// TIA Portal V15.1 export
// export: Created 2024-06-21T08:41:06.2222492Z, ExportSetting WithDefaults, DisplayName Totally Integrated Automation Portal, DisplayVersion V15.1 Update 5, DisplayName TIA Portal Openness, DisplayVersion V15.1 Update 5, DisplayName SINAMICS Startdrive Advanced, DisplayVersion V15.1, DisplayName G130, G150, S120, S150, SINAMICS MV, S210, DisplayVersion V15.1, DisplayName G110M, G120, G120C, G120D, G120P, DisplayVersion V15.1, DisplayName STEP 7 Professional, DisplayVersion V15.1 Update 5, DisplayName STEP 7 Safety, DisplayVersion V15.1, DisplayName WinCC Professional, DisplayVersion V15.1 Update 5, DisplayName SIMATIC Visualization Architect, DisplayVersion V15.1
FUNCTION_BLOCK "LGBMotorEPos-MoviProPN"   // FB6622, FBD
TITLE = LMotorMovUnitEPos-MoviProPN / LGBMotorEPos-MoviProPN
{ S7_Optimized_Access := 'TRUE' }
VERSION : 0.1
// ============================================================================
// This module is used in applications when a Motor positioning equipped with SEW MOVIPRO with fieldbus steering is needed.
// ============================================================================
// stored: AutoNumber false, IsIECCheckEnabled false, IsRetainMemResEnabled false, MemoryReserve 100, SetENOAutomatically False, UDAEnableTagReadback false
   VAR_INPUT
      I_MotorProtection { ExternalAccessible := 'False'; ExternalVisible := 'False'; ExternalWritable := 'False'} : Bool;   // Motor protection
      I_AlarmResetPB { ExternalAccessible := 'False'; ExternalVisible := 'False'; ExternalWritable := 'False'} : Bool;   // Alarm Reset Pushbutton is Activated
      I_SafetyStatusWord { ExternalAccessible := 'False'; ExternalVisible := 'False'; ExternalWritable := 'False'} : Word;   // Safety status word
      I_SafetyControlWord { ExternalAccessible := 'False'; ExternalVisible := 'False'; ExternalWritable := 'False'} : Word;   // Safety control word
      I_SafetyOk { ExternalAccessible := 'False'; ExternalVisible := 'False'; ExternalWritable := 'False'} : Bool;   // Safety ok
      I_MotionStopOk { ExternalAccessible := 'False'; ExternalVisible := 'False'; ExternalWritable := 'False'} : Bool;   // Safety Ok / The motion stop is Ok
      I_ContolInhibit { ExternalAccessible := 'False'; ExternalVisible := 'False'; ExternalWritable := 'False'} : Bool;   // Inhibit motor (disable output stage, uncontolled stop)
      I_Start { ExternalAccessible := 'False'; ExternalVisible := 'False'; ExternalWritable := 'False'} : Bool;
      I_OFF2 { ExternalAccessible := 'False'; ExternalVisible := 'False'; ExternalWritable := 'False'} : Bool := True;   // OFF2 rapid stop
      I_SetpointPosition { ExternalAccessible := 'False'; ExternalVisible := 'False'; ExternalWritable := 'False'} : DInt;   // Setpoint position [ user unit ex: rev. ]
      I_SetpointSpeed { ExternalAccessible := 'False'; ExternalVisible := 'False'; ExternalWritable := 'False'} : Int;   // Setpoint velocity [ user unit ex: rev./min ]
      I_Acceleration { ExternalAccessible := 'False'; ExternalVisible := 'False'; ExternalWritable := 'False'} : Int;   // Acceleration [ user unit ex: rev./(min*S) ]
      I_Deceleration { ExternalAccessible := 'False'; ExternalVisible := 'False'; ExternalWritable := 'False'} : Int;   // Deceleration [ user unit ex: rev./(min*S) ]
      I_OperatingMode { ExternalAccessible := 'False'; ExternalVisible := 'False'; ExternalWritable := 'False'} : USInt := 4;   // 0=Default, 1=Speed control, 2=Jog mode, 3=Referencing mode, 4=Positioning mode, 5=Positioning mode - touch probe, 6=Speed synchronization, 7=Emergency mode
      I_BrakeRelease { ExternalAccessible := 'False'; ExternalVisible := 'False'; ExternalWritable := 'False'} : Bool;   // Command brake release
      I_DisableSoftwareLimitSwitches { ExternalAccessible := 'False'; ExternalVisible := 'False'; ExternalWritable := 'False'} : Bool;   // Disable softwrare limit switches in the drive
      I_EnableTorqueLimiting { ExternalAccessible := 'False'; ExternalVisible := 'False'; ExternalWritable := 'False'} : Bool;   // Enable torque limiting
      I_JogPositive { ExternalAccessible := 'False'; ExternalVisible := 'False'; ExternalWritable := 'False'} : Bool;   // Jog in positive direction
      I_JogNegative { ExternalAccessible := 'False'; ExternalVisible := 'False'; ExternalWritable := 'False'} : Bool;   // Jog in negative direction
   END_VAR
   VAR_OUTPUT
      O_MotorProtectionAlarm { ExternalAccessible := 'False'; ExternalVisible := 'False'; ExternalWritable := 'False'} : Bool;   // Motor protection alarm
      O_SafetySwitchAlarm { ExternalAccessible := 'False'; ExternalVisible := 'False'; ExternalWritable := 'False'} : Bool;   // Safety switch alarm
      O_STOAlarm { ExternalAccessible := 'False'; ExternalVisible := 'False'; ExternalWritable := 'False'} : Bool;   // Drive fault / STO alarm
      O_MotionStopWarning { ExternalAccessible := 'False'; ExternalVisible := 'False'; ExternalWritable := 'False'} : Bool;   // Drive fault / Motion Stop warning
      O_DriveFaultAlarm { ExternalAccessible := 'False'; ExternalVisible := 'False'; ExternalWritable := 'False'} : Bool;   // Drive fault
      O_DriveWarning { ExternalAccessible := 'False'; ExternalVisible := 'False'; ExternalWritable := 'False'} : Bool;   // Drive warning
      O_DriveReady { ExternalAccessible := 'False'; ExternalVisible := 'False'; ExternalWritable := 'False'} : Bool;   // Drive ready
      O_Referenced { ExternalAccessible := 'False'; ExternalVisible := 'False'; ExternalWritable := 'False'} : Bool;   // Drive is referenced
      O_MotorTurning { ExternalAccessible := 'False'; ExternalVisible := 'False'; ExternalWritable := 'False'} : Bool;   // Inverter output stage is enabled
      O_Brake { ExternalAccessible := 'False'; ExternalVisible := 'False'; ExternalWritable := 'False'} : Bool;   // Brake status
      O_Standstill { ExternalAccessible := 'False'; ExternalVisible := 'False'; ExternalWritable := 'False'} : Bool;   // Sandstill
      O_SetpointReached { ExternalAccessible := 'False'; ExternalVisible := 'False'; ExternalWritable := 'False'} : Bool;   // Setpoint position is reached
      O_HWLSPositive { ExternalAccessible := 'False'; ExternalVisible := 'False'; ExternalWritable := 'False'} : Bool;   // Hardware limit switch positive reached
      O_HWLSNegative { ExternalAccessible := 'False'; ExternalVisible := 'False'; ExternalWritable := 'False'} : Bool;   // Hardware limit switch negative reached
      O_NoResponse { ExternalAccessible := 'False'; ExternalVisible := 'False'; ExternalWritable := 'False'} : Bool;   // No response / O_NoResponse
      O_ActualPosition { ExternalAccessible := 'False'; ExternalVisible := 'False'; ExternalWritable := 'False'} : DInt;   // Actual position
      O_AlarmABCondition { ExternalAccessible := 'False'; ExternalVisible := 'False'; ExternalWritable := 'False'} : Bool;   // Alarm AB Condition
      H_IAnim { ExternalAccessible := 'False'; ExternalVisible := 'False'; ExternalWritable := 'False'} : DWord;   // Icon Animation
   END_VAR
   VAR_IN_OUT
      IO_Alarm : "Alarm";
      "H_GBMotorEPos-MoviProPN" : "H_GBMotorEPos-MoviProPN";   // HMI UDT
      C_EnableAlarm { ExternalAccessible := 'False'; ExternalVisible := 'False'; ExternalWritable := 'False'} : Bool;   // Enable Alarm
      C_MotorProtectionUsed { ExternalAccessible := 'False'; ExternalVisible := 'False'; ExternalWritable := 'False'} : Bool := True;   // Motor Protection used
      C_MotorProtectionNc { ExternalAccessible := 'False'; ExternalVisible := 'False'; ExternalWritable := 'False'} : Bool := True;   // Motor Protection Normally closed
      C_MotionStopUsed { ExternalAccessible := 'False'; ExternalVisible := 'False'; ExternalWritable := 'False'} : Bool;   // Motion Stop used
      C_HWSubInput { ExternalAccessible := 'False'; ExternalVisible := 'False'; ExternalWritable := 'False'} : HW_SUBMODULE;   // Inputs telegram 3 Hardware identifier
      C_HWSubOutput { ExternalAccessible := 'False'; ExternalVisible := 'False'; ExternalWritable := 'False'} : HW_SUBMODULE;   // Outputs telegram 3 Hardware identifier
      C_HWSubControllerInput { ExternalAccessible := 'False'; ExternalVisible := 'False'; ExternalWritable := 'False'} : HW_SUBMODULE;   // Controller inputs telegram 2 Hardware identifier
      C_HWSubControllerOutput { ExternalAccessible := 'False'; ExternalVisible := 'False'; ExternalWritable := 'False'} : HW_SUBMODULE;   // Controller outputs telegram 2 Hardware identifier
      C_DriveCurrent { ExternalAccessible := 'False'; ExternalVisible := 'False'; ExternalWritable := 'False'} : Real;   // Reference current of the drive
      C_MotorCurrent { ExternalAccessible := 'False'; ExternalVisible := 'False'; ExternalWritable := 'False'} : Real;   // Reference current of the motor
   END_VAR
   VAR
      MotorProtectionAlarm { ExternalAccessible := 'False'; ExternalVisible := 'False'; ExternalWritable := 'False'} : Bool;   // Motor protection alarm
      MotorProtectionAlarmABCond { ExternalAccessible := 'False'; ExternalVisible := 'False'; ExternalWritable := 'False'} : Bool;   // Motor protection alarm condition
      SafetySwitchAlarm { ExternalAccessible := 'False'; ExternalVisible := 'False'; ExternalWritable := 'False'} : Bool;   // Safety Switch alarm
      SafetySwitchAlarmABCond { ExternalAccessible := 'False'; ExternalVisible := 'False'; ExternalWritable := 'False'} : Bool;   // Safety Switch alarm condition
      DriveFaultAlarm { ExternalAccessible := 'False'; ExternalVisible := 'False'; ExternalWritable := 'False'} : Bool;   // Drive fault alarm
      DriveFaultAlarmABCond { ExternalAccessible := 'False'; ExternalVisible := 'False'; ExternalWritable := 'False'} : Bool;   // Drive fault alarm condition
      STOAlarm { ExternalAccessible := 'False'; ExternalVisible := 'False'; ExternalWritable := 'False'} : Bool;   // Drive fault alarm / STO feedback fault alarm
      STOAlarmABCond { ExternalAccessible := 'False'; ExternalVisible := 'False'; ExternalWritable := 'False'} : Bool;   // Drive fault alarm condition / STO feedback fault alarm condition
      MotionStopWarning { ExternalAccessible := 'False'; ExternalVisible := 'False'; ExternalWritable := 'False'} : Bool;   // Drive fault alarm / Motion Stop warning
      Start { ExternalAccessible := 'False'; ExternalVisible := 'False'; ExternalWritable := 'False'} : Bool;   // Start command to drive
      MotorTurning { ExternalAccessible := 'False'; ExternalVisible := 'False'; ExternalWritable := 'False'} : Bool;   // Motor is turning
      MaintenanceSwitch { ExternalAccessible := 'False'; ExternalVisible := 'False'; ExternalWritable := 'False'} : Bool;   // Maintenance switch activated (1=mains OFF)
      Fault { ExternalAccessible := 'False'; ExternalVisible := 'False'; ExternalWritable := 'False'} : Bool;   // Fault present
      Warning { ExternalAccessible := 'False'; ExternalVisible := 'False'; ExternalWritable := 'False'} : Bool;   // Warning present
      ApplicationFault { ExternalAccessible := 'False'; ExternalVisible := 'False'; ExternalWritable := 'False'} : Bool;   // Application fault present
      Brake { ExternalAccessible := 'False'; ExternalVisible := 'False'; ExternalWritable := 'False'} : Bool;   // Brake status
      AliveBit { ExternalAccessible := 'False'; ExternalVisible := 'False'; ExternalWritable := 'False'} : Bool;   // Toggles default every 100ms
      AliveBitOffDlyOk { ExternalAccessible := 'False'; ExternalVisible := 'False'; ExternalWritable := 'False'} : Bool;
      AliveBitOnDlyOk { ExternalAccessible := 'False'; ExternalVisible := 'False'; ExternalWritable := 'False'} : Bool;
      AliveBitStatusOk { ExternalAccessible := 'False'; ExternalVisible := 'False'; ExternalWritable := 'False'} : Bool;
      _MoviproPN { ExternalAccessible := 'False'; ExternalVisible := 'False'; ExternalWritable := 'False'} : "LGBSEW-MoviProPN";   // SEW MOVIFIT FC
      _MotorProtection { ExternalAccessible := 'False'; ExternalVisible := 'False'; ExternalWritable := 'False'} : "L1AlarmMultiIn";   // FB
      _SafetySwitch { ExternalAccessible := 'False'; ExternalVisible := 'False'; ExternalWritable := 'False'} : "L1AlarmMultiIn";   // FB
      _DriveFault { ExternalAccessible := 'False'; ExternalVisible := 'False'; ExternalWritable := 'False'} : "L1AlarmMultiIn";   // FB
      _STO { ExternalAccessible := 'False'; ExternalVisible := 'False'; ExternalWritable := 'False'} : "L1AlarmMultiIn";   // FB
      _MotionStop { ExternalAccessible := 'False'; ExternalVisible := 'False'; ExternalWritable := 'False'} : "L1AlarmMultiIn";   // FB
      T_STOAlarm { ExternalAccessible := 'False'; ExternalVisible := 'False'; ExternalWritable := 'False'} : TON_TIME;   // Timer
      T_AliveBitOnDly { ExternalAccessible := 'False'; ExternalVisible := 'False'; ExternalWritable := 'False'} : TON_TIME;   // Timer
      T_AliveBitOffDly { ExternalAccessible := 'False'; ExternalVisible := 'False'; ExternalWritable := 'False'} : TOF_TIME;   // Timer
   END_VAR
BEGIN

REGION Network 1: **** 2.2 - Alarms - Alarm Generation **** Motor Protection Alarm
   // Motor Protection Alarm
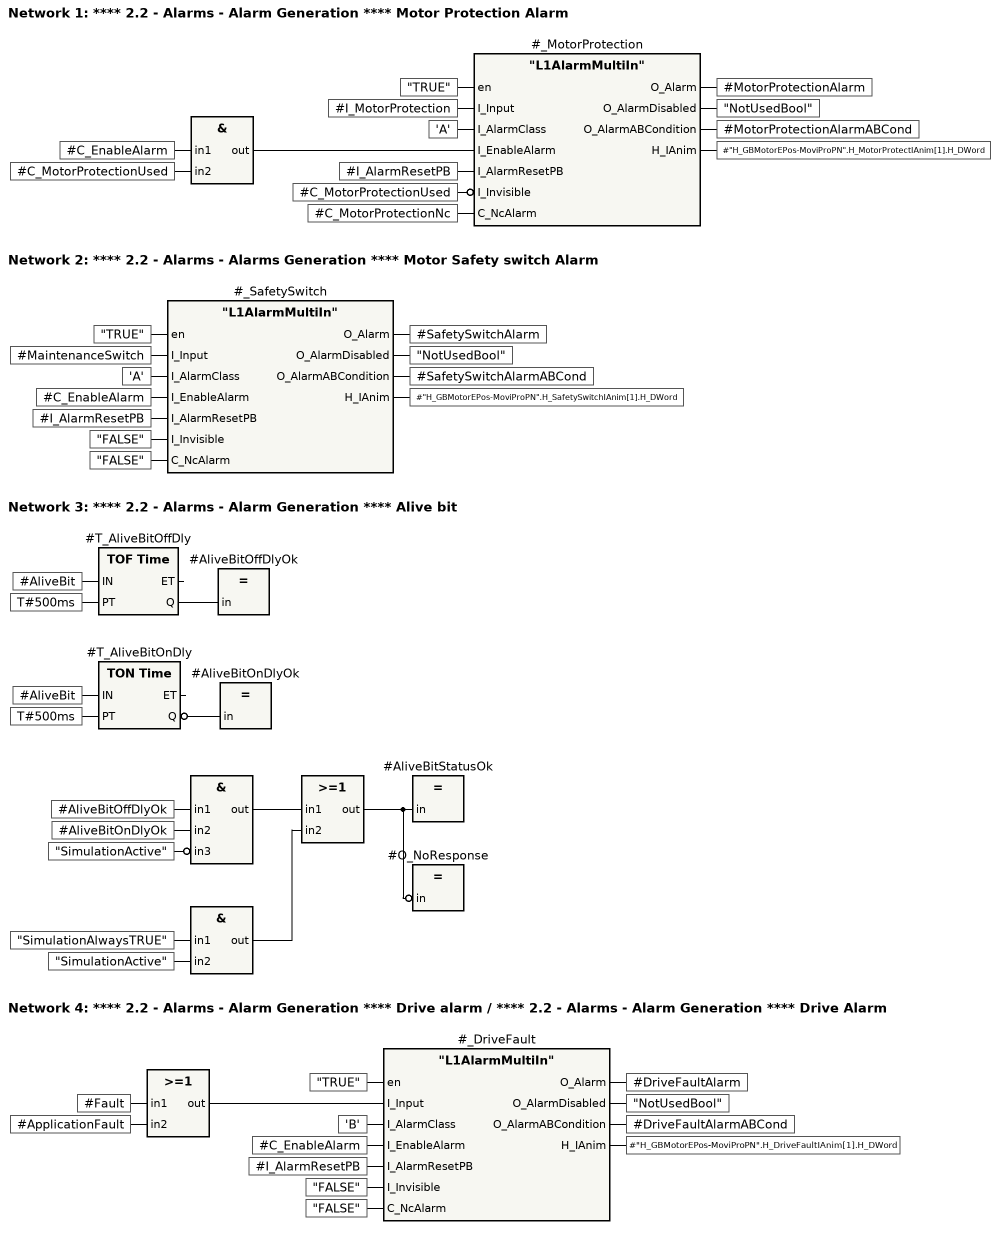
   IF "TRUE" THEN
       #_MotorProtection(I_Input := #I_MotorProtection,   // "L1AlarmMultiIn"
                         I_AlarmClass := 'A',
                         I_EnableAlarm := #C_EnableAlarm AND #C_MotorProtectionUsed,
                         I_AlarmResetPB := #I_AlarmResetPB,
                         I_Invisible := NOT #C_MotorProtectionUsed,
                         C_NcAlarm := #C_MotorProtectionNc,
                         O_Alarm => #MotorProtectionAlarm,
                         O_AlarmDisabled => "NotUsedBool",
                         O_AlarmABCondition => #MotorProtectionAlarmABCond,
                         H_IAnim => #"H_GBMotorEPos-MoviProPN".H_MotorProtectIAnim[1].H_DWord);
   END_IF;
END_REGION

REGION Network 2: **** 2.2 - Alarms - Alarms Generation **** Motor Safety switch Alarm
   // Motor Safety switch Alarm
   IF "TRUE" THEN
       #_SafetySwitch(I_Input := #MaintenanceSwitch,   // "L1AlarmMultiIn"
                      I_AlarmClass := 'A',
                      I_EnableAlarm := #C_EnableAlarm,
                      I_AlarmResetPB := #I_AlarmResetPB,
                      I_Invisible := "FALSE",
                      C_NcAlarm := "FALSE",
                      O_Alarm => #SafetySwitchAlarm,
                      O_AlarmDisabled => "NotUsedBool",
                      O_AlarmABCondition => #SafetySwitchAlarmABCond,
                      H_IAnim => #"H_GBMotorEPos-MoviProPN".H_SafetySwitchIAnim[1].H_DWord);
   END_IF;
END_REGION

REGION Network 3: **** 2.2 - Alarms - Alarm Generation **** Alive bit
   #T_AliveBitOffDly(IN := #AliveBit, PT := T#500ms);   // TOF
   #AliveBitOffDlyOk := #T_AliveBitOffDly.Q;   // ^ Start of Off delay l _ / _ _ l_l l__________l l__l l_______ l------------------\--------------------------------------> t (s) \ more then 500ms have passed without a "True" signal. Status is set to NOK, an error is generated.
   #T_AliveBitOnDly(IN := #AliveBit, PT := T#500ms);   // TON
   #AliveBitOnDlyOk := NOT #T_AliveBitOnDly.Q;   // ^ Start of On delay l _ /_______ _ _ l_l l__l \ l____l l__l l_______ l------------------\--------------------------------------> t (s) \ more then 500ms have passed without a "False" signal. Status is set to NOK, an error is generated.
   #AliveBitStatusOk := (#AliveBitOffDlyOk AND #AliveBitOnDlyOk AND NOT "SimulationActive") OR ("SimulationAlwaysTRUE" AND "SimulationActive");   // On and off pulse are each 100ms in normal operation. ^ l _ _ _ _ _ _ _ the satus is OK l_l l__l l__l l__l l__l l__l l__l l l--------------------------------------------------------> t (s)
   #O_NoResponse := NOT #AliveBitStatusOk;
END_REGION

REGION Network 4: **** 2.2 - Alarms - Alarm Generation **** Drive alarm / **** 2.2 - Alarms - Alarm Generation **** Drive Alarm
   IF "TRUE" THEN
       #_DriveFault(I_Input := #Fault OR #ApplicationFault,   // "L1AlarmMultiIn"
                    I_AlarmClass := 'B',
                    I_EnableAlarm := #C_EnableAlarm,
                    I_AlarmResetPB := #I_AlarmResetPB,
                    I_Invisible := "FALSE",
                    C_NcAlarm := "FALSE",
                    O_Alarm => #DriveFaultAlarm,
                    O_AlarmDisabled => "NotUsedBool",
                    O_AlarmABCondition => #DriveFaultAlarmABCond,
                    H_IAnim => #"H_GBMotorEPos-MoviProPN".H_DriveFaultIAnim[1].H_DWord);
   END_IF;
END_REGION

REGION Network 5: **** 2.2 - Alarms - Alarm Generation **** STO Alarm
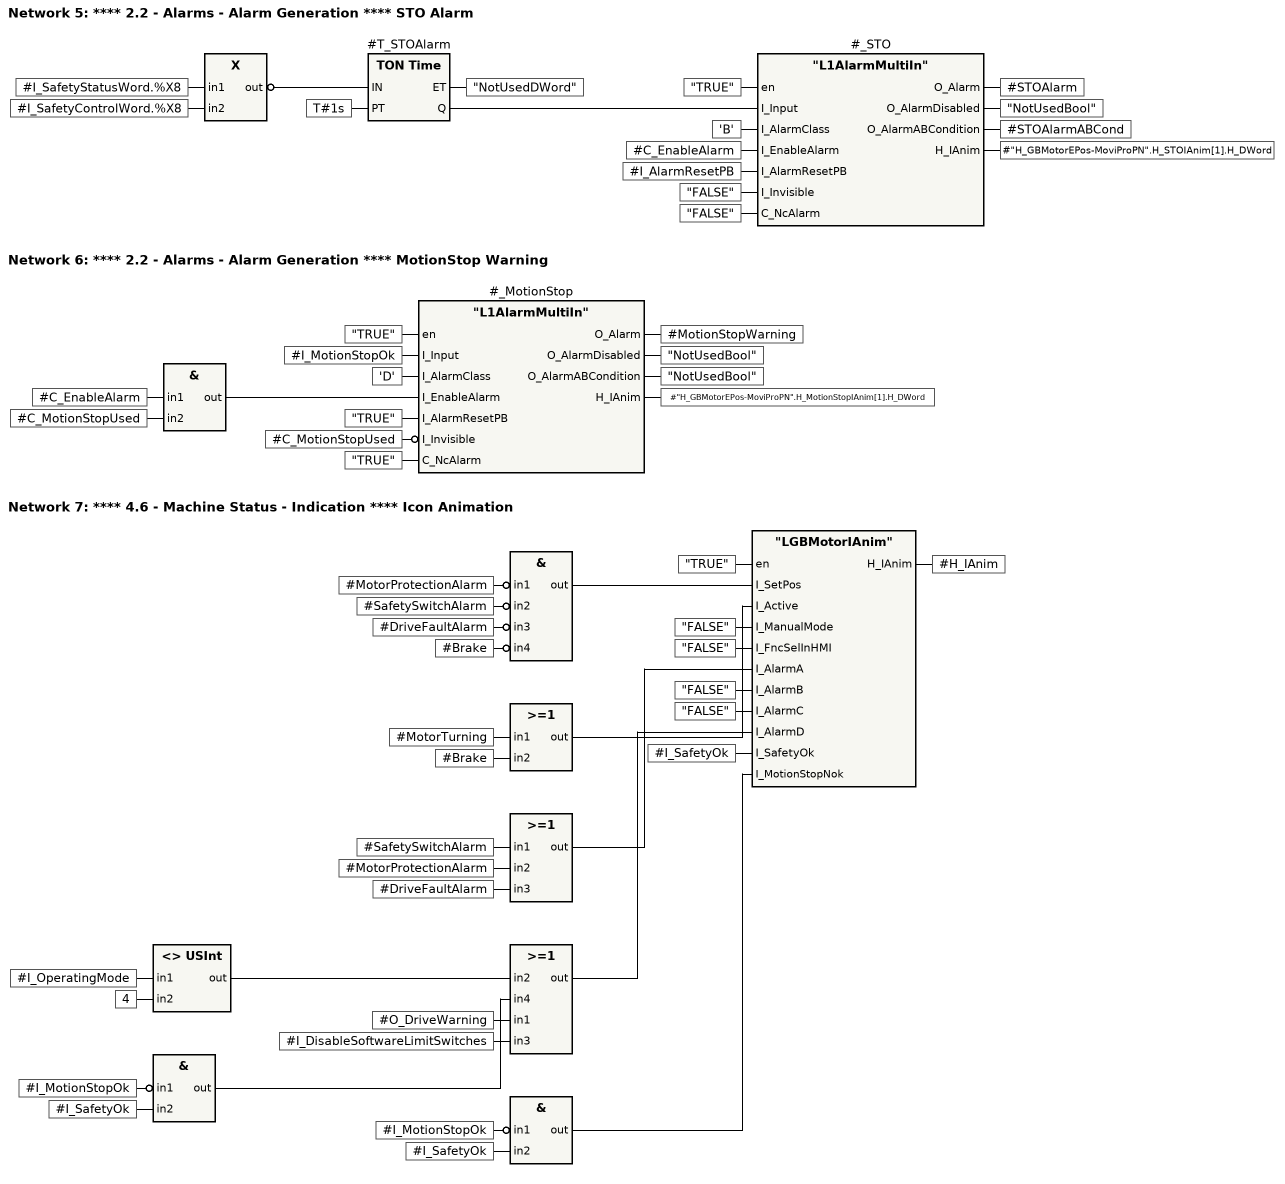
   #T_STOAlarm(IN := NOT (#I_SafetyStatusWord.%X8 XOR #I_SafetyControlWord.%X8),   // TON
               PT := T#1s,
               ET => "NotUsedDWord");
   IF "TRUE" THEN
       #_STO(I_Input := #T_STOAlarm.Q,   // "L1AlarmMultiIn"
             I_AlarmClass := 'B',
             I_EnableAlarm := #C_EnableAlarm,
             I_AlarmResetPB := #I_AlarmResetPB,
             I_Invisible := "FALSE",
             C_NcAlarm := "FALSE",
             O_Alarm => #STOAlarm,
             O_AlarmDisabled => "NotUsedBool",
             O_AlarmABCondition => #STOAlarmABCond,
             H_IAnim => #"H_GBMotorEPos-MoviProPN".H_STOIAnim[1].H_DWord);
   END_IF;
END_REGION

REGION Network 6: **** 2.2 - Alarms - Alarm Generation **** MotionStop Warning
   IF "TRUE" THEN
       #_MotionStop(I_Input := #I_MotionStopOk,   // "L1AlarmMultiIn"
                    I_AlarmClass := 'D',
                    I_EnableAlarm := #C_EnableAlarm AND #C_MotionStopUsed,
                    I_AlarmResetPB := "TRUE",
                    I_Invisible := NOT #C_MotionStopUsed,
                    C_NcAlarm := "TRUE",
                    O_Alarm => #MotionStopWarning,
                    O_AlarmDisabled => "NotUsedBool",
                    O_AlarmABCondition => "NotUsedBool",
                    H_IAnim => #"H_GBMotorEPos-MoviProPN".H_MotionStopIAnim[1].H_DWord);
   END_IF;
END_REGION

REGION Network 7: **** 4.6 - Machine Status - Indication **** Icon Animation
   // Icon Animation
   IF "TRUE" THEN
       "LGBMotorIAnim"(I_SetPos := NOT #MotorProtectionAlarm AND NOT #SafetySwitchAlarm AND NOT #DriveFaultAlarm AND NOT #Brake,
                       I_Active := #MotorTurning OR #Brake,
                       I_ManualMode := "FALSE",
                       I_FncSelInHMI := "FALSE",
                       I_AlarmA := #SafetySwitchAlarm OR #MotorProtectionAlarm OR #DriveFaultAlarm,
                       I_AlarmB := "FALSE",
                       I_AlarmC := "FALSE",
                       I_AlarmD := (#I_OperatingMode <> 4) OR (NOT #I_MotionStopOk AND #I_SafetyOk) OR #O_DriveWarning OR #I_DisableSoftwareLimitSwitches,
                       I_SafetyOk := #I_SafetyOk,
                       I_MotionStopNok := NOT #I_MotionStopOk AND #I_SafetyOk,
                       H_IAnim => #H_IAnim);
   END_IF;
END_REGION

REGION Network 8: **** 4.6 - Machine Status - Indication **** Animation
   // Animation
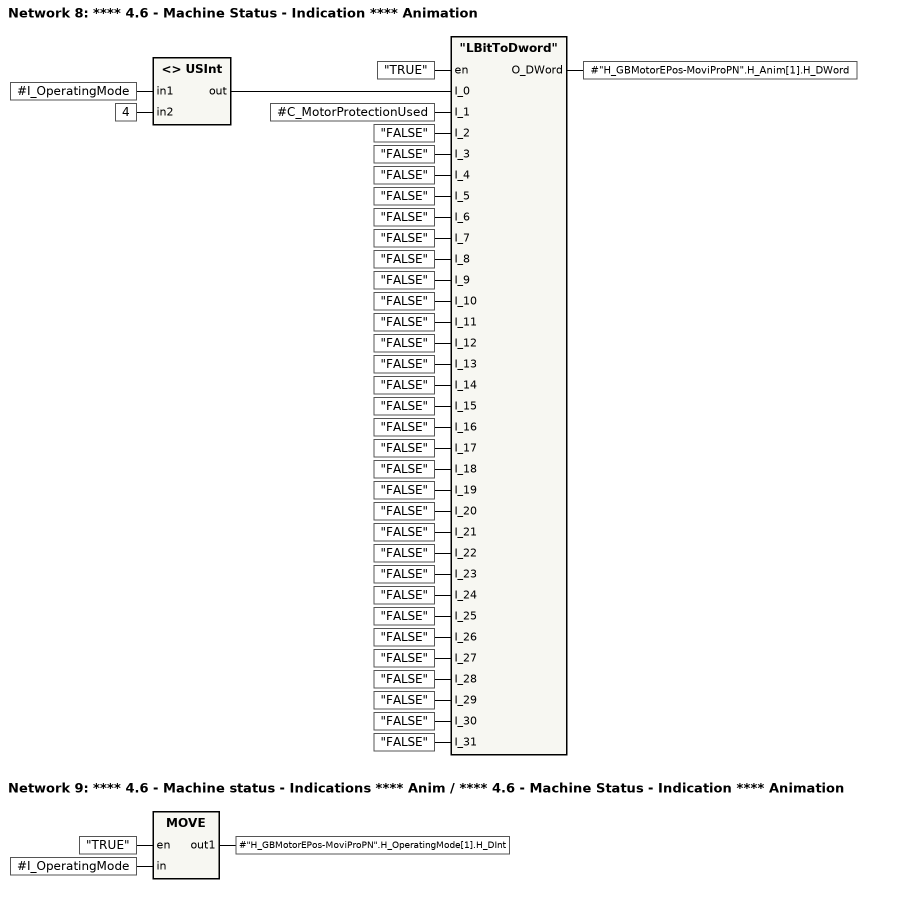
   IF "TRUE" THEN
       "LBitToDword"(I_0 := #I_OperatingMode <> 4,   // HMI PLC __________________________________________________________ l _SIEMENS____________________________SIMATIC HMI_____ l ___________________ l l l l l_l_l_l______________l l l l l l SIEMENS SIMATIC l l l ________________ l l l ________S7-1500 l l l l_____________ X l l l l l___________O_l l l l l l l l l l l l l l l Popup or l l l l l l l l l l screen. l l l l l l l l l l l <<-------==================l= l========= l l l l l l l Anim l l l l l______________l l l l l_______________l l l l ___ l l l l l l __l l__ l l l l l l l__ __l l l l l l l l___l l l l l l l l l l_____________________________________________________ l l l__________________ l l_________________________________________________________ l Animation word is send to the HMI to be used in object screen or popup _
                     I_1 := #C_MotorProtectionUsed,
                     I_2 := "FALSE",
                     I_3 := "FALSE",
                     I_4 := "FALSE",
                     I_5 := "FALSE",
                     I_6 := "FALSE",
                     I_7 := "FALSE",
                     I_8 := "FALSE",
                     I_9 := "FALSE",
                     I_10 := "FALSE",
                     I_11 := "FALSE",
                     I_12 := "FALSE",
                     I_13 := "FALSE",
                     I_14 := "FALSE",
                     I_15 := "FALSE",
                     I_16 := "FALSE",
                     I_17 := "FALSE",
                     I_18 := "FALSE",
                     I_19 := "FALSE",
                     I_20 := "FALSE",
                     I_21 := "FALSE",
                     I_22 := "FALSE",
                     I_23 := "FALSE",
                     I_24 := "FALSE",
                     I_25 := "FALSE",
                     I_26 := "FALSE",
                     I_27 := "FALSE",
                     I_28 := "FALSE",
                     I_29 := "FALSE",
                     I_30 := "FALSE",
                     I_31 := "FALSE",
                     O_DWord => #"H_GBMotorEPos-MoviProPN".H_Anim[1].H_DWord);
   END_IF;
END_REGION

REGION Network 9: **** 4.6 - Machine status - Indications **** Anim / **** 4.6 - Machine Status - Indication **** Animation
   // Anim
   IF "TRUE" THEN
       #"H_GBMotorEPos-MoviProPN".H_OperatingMode[1].H_DInt := #I_OperatingMode;   // HMI PLC __________________________________________________________ l _SIEMENS____________________________SIMATIC HMI_____ l ___________________ l l l l l_l_l_l______________l l l l l l SIEMENS SIMATIC l l l ________________ l l l ________S7-1500 l l l l_____________ X l l l l l___________O_l l l l l l l l l l l l l l l Popup or l l l l l l l l l l screen. l l l l l l l l l l l <<-------==================l= l========= l l l l l l l Anim l l l l l______________l l l l l_______________l l l l ___ l l l l l l __l l__ l l l l l l l__ __l l l l l l l l___l l l l l l l l l l_____________________________________________________ l l l__________________ l l_________________________________________________________ l Animation word is send to the HMI to be used in object screen or popup _
   END_IF;
END_REGION

REGION Network 10: **** 4.6 - Machine Status - Indication **** Safety words
   // Animation
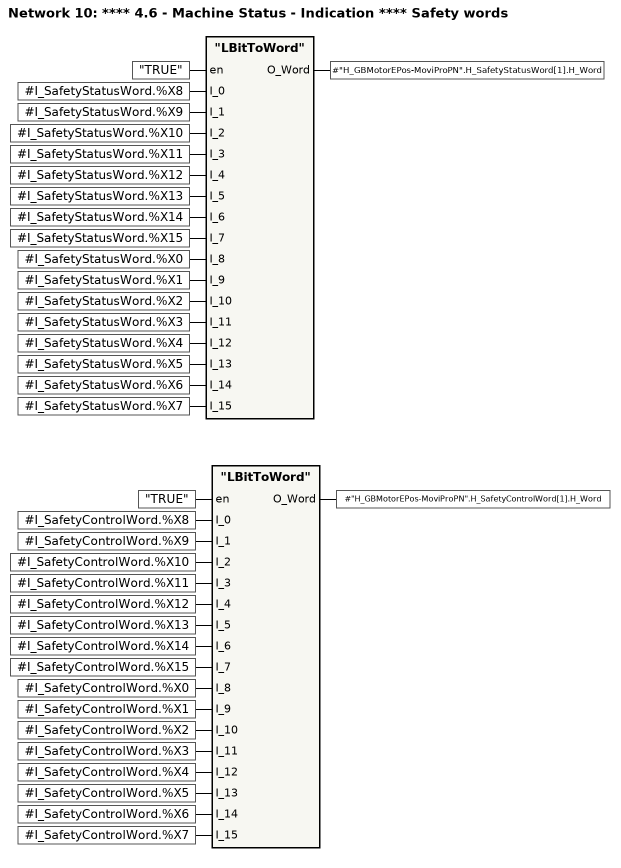
   IF "TRUE" THEN
       "LBitToWord"(I_0 := #I_SafetyStatusWord.%X8,
                    I_1 := #I_SafetyStatusWord.%X9,
                    I_2 := #I_SafetyStatusWord.%X10,
                    I_3 := #I_SafetyStatusWord.%X11,
                    I_4 := #I_SafetyStatusWord.%X12,
                    I_5 := #I_SafetyStatusWord.%X13,
                    I_6 := #I_SafetyStatusWord.%X14,
                    I_7 := #I_SafetyStatusWord.%X15,
                    I_8 := #I_SafetyStatusWord.%X0,
                    I_9 := #I_SafetyStatusWord.%X1,
                    I_10 := #I_SafetyStatusWord.%X2,
                    I_11 := #I_SafetyStatusWord.%X3,
                    I_12 := #I_SafetyStatusWord.%X4,
                    I_13 := #I_SafetyStatusWord.%X5,
                    I_14 := #I_SafetyStatusWord.%X6,
                    I_15 := #I_SafetyStatusWord.%X7,
                    O_Word => #"H_GBMotorEPos-MoviProPN".H_SafetyStatusWord[1].H_Word);
   END_IF;
   IF "TRUE" THEN
       "LBitToWord"(I_0 := #I_SafetyControlWord.%X8,
                    I_1 := #I_SafetyControlWord.%X9,
                    I_2 := #I_SafetyControlWord.%X10,
                    I_3 := #I_SafetyControlWord.%X11,
                    I_4 := #I_SafetyControlWord.%X12,
                    I_5 := #I_SafetyControlWord.%X13,
                    I_6 := #I_SafetyControlWord.%X14,
                    I_7 := #I_SafetyControlWord.%X15,
                    I_8 := #I_SafetyControlWord.%X0,
                    I_9 := #I_SafetyControlWord.%X1,
                    I_10 := #I_SafetyControlWord.%X2,
                    I_11 := #I_SafetyControlWord.%X3,
                    I_12 := #I_SafetyControlWord.%X4,
                    I_13 := #I_SafetyControlWord.%X5,
                    I_14 := #I_SafetyControlWord.%X6,
                    I_15 := #I_SafetyControlWord.%X7,
                    O_Word => #"H_GBMotorEPos-MoviProPN".H_SafetyControlWord[1].H_Word);
   END_IF;
END_REGION

REGION Network 11: **** 7.3 - Submodule - Machine **** MoviPro
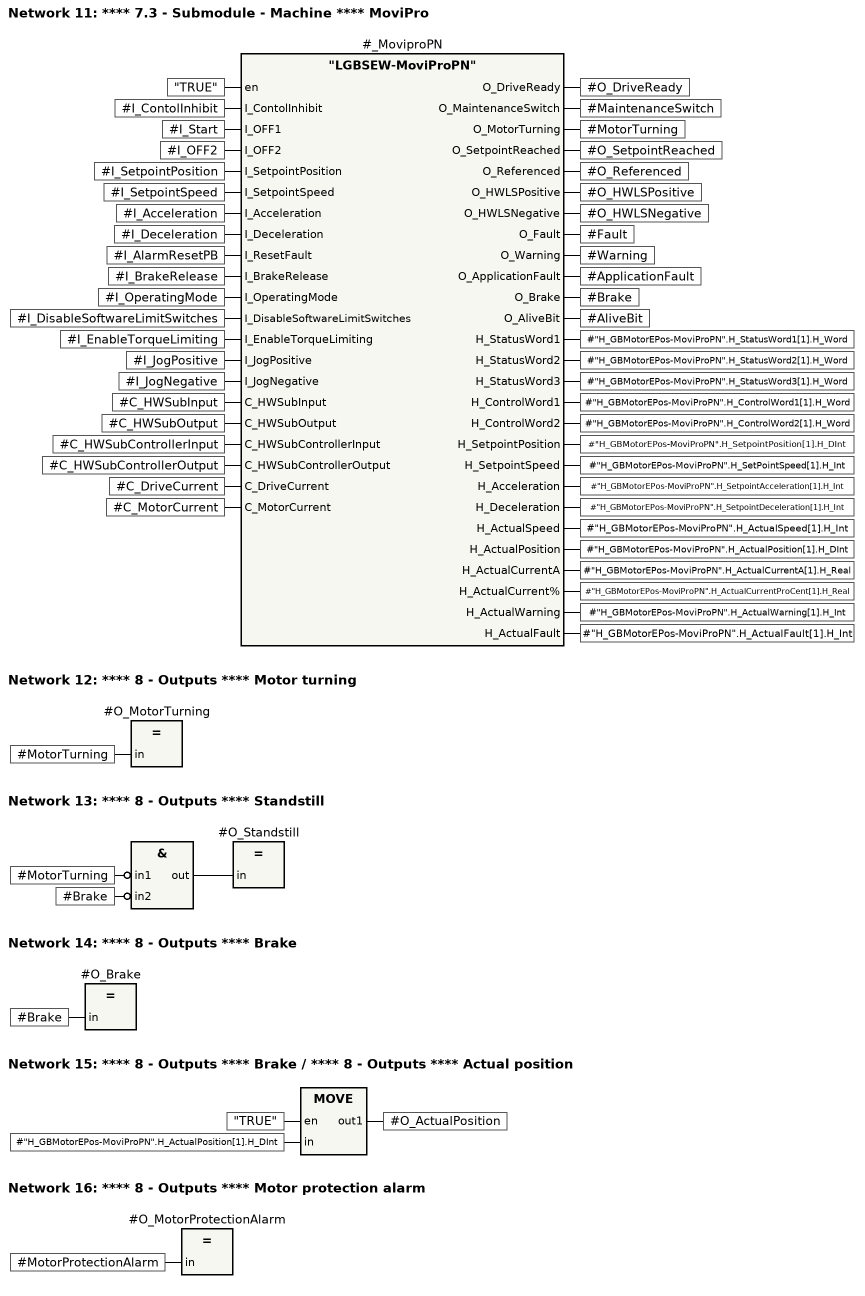
   IF "TRUE" THEN
       #_MoviproPN(I_ContolInhibit := #I_ContolInhibit,   // "LGBSEW-MoviProPN": Quick stop "I_OFF2" : ^ Speed (%) Stop signal at 5s l / 100% l______________/_ l \ \ l \ \ l \ \ l \ \ 0% l___________________\_____\___________________________> Time (s) l OFF2 OFF1 (regular start stop) 7s 10s ************************************************************************************ "I_SetpointSpeed" , "I_Acceleration", "I_Deceleration": Speed Target speed (user unit) ^ / l ____/____ l / \ l / \ l____/ \____ l--------------------------------------------------> t (s) Speed (user unit) ^ Acceleration l l _________ l l / \ l l/ \ l____/ \____ l--------------------------------------------------> t (s) Speed (user unit) ^ Deceleration l _________ l l / \ l l / \l l____/ \____ l--------------------------------------------------> t (s) ************************************************************************************ Mode selection bits "I_OperatingMode" : mode: 0=Default 1=Speed control 2=Jog mode 3=Referencing mode 4=Positioning mode 5=Positioning mode - touch probe 6=Speed synchronization 7=Emergency mode ************************************************************************************ Software limit switches "I_DisbaleSoftwareLimitSwitches" : The software limit switches are programmed before the hardware limit switches. This will give the drive the possiblility to decelarate accordingly as its knows the distance to these SW LS's from the encoder value. When the referencing is ok it should be impossible to reach the hardware limit switches. Only when there is a faulty referencing then the software limit switches can be behind the hardware limit switch. In that case it is possible to hit the hardware limit switch with full speed. Positive <-- Load --> negative HW LS SW LS _____ SW LS HW LS ____ ____ l_____l ____ ____ l____\ l____\ l_____l /____l /____l OOOOOOOOOOOOOOOOOOOOOOOOOOOOOOOOOOOO ll // \\ ll ll// \\ll ll ll ************************************************************************************ Input "I_EnableTorqueLimiting" : 110% ^ Torque (%) l Torque limited 100% l_______________________________/___________________ torque limit configured in the drive l _ Acceleration l l l l l / l l---- shutdown command l l l/ constant speed l l (error motor blocked) l l l_____/__ l l 0% l___l_________l________________l__l___________________________> Time (s) l l l l l l l / l l l / l_l -100% l __________ /________________________________________ torque limit configured in the drive l Deceleration -110% l ************************************************************************************ Communication handeling is done in the block with the "C_HWSub..." hardware identifiers. SEW Drive ______________ ll __ _ ll__ input telegram ll l__l l_l ll Ol ===============>> PLC ll ll__l ll_____________ll l__l l__l l_ll_l SEW Drive ______________ output telegram ll __ _ ll__ PLC ===============>> ll l__l l_l ll Ol ll ll__l ll_____________ll l__l l__l l_ll_l _
                   I_OFF1 := #I_Start,
                   I_OFF2 := #I_OFF2,
                   I_SetpointPosition := #I_SetpointPosition,
                   I_SetpointSpeed := #I_SetpointSpeed,
                   I_Acceleration := #I_Acceleration,
                   I_Deceleration := #I_Deceleration,
                   I_ResetFault := #I_AlarmResetPB,
                   I_BrakeRelease := #I_BrakeRelease,
                   I_OperatingMode := #I_OperatingMode,
                   I_DisableSoftwareLimitSwitches := #I_DisableSoftwareLimitSwitches,
                   I_EnableTorqueLimiting := #I_EnableTorqueLimiting,
                   I_JogPositive := #I_JogPositive,
                   I_JogNegative := #I_JogNegative,
                   C_HWSubInput := #C_HWSubInput,
                   C_HWSubOutput := #C_HWSubOutput,
                   C_HWSubControllerInput := #C_HWSubControllerInput,
                   C_HWSubControllerOutput := #C_HWSubControllerOutput,
                   C_DriveCurrent := #C_DriveCurrent,
                   C_MotorCurrent := #C_MotorCurrent,
                   O_DriveReady => #O_DriveReady,
                   O_MaintenanceSwitch => #MaintenanceSwitch,
                   O_MotorTurning => #MotorTurning,
                   O_SetpointReached => #O_SetpointReached,
                   O_Referenced => #O_Referenced,
                   O_HWLSPositive => #O_HWLSPositive,
                   O_HWLSNegative => #O_HWLSNegative,
                   O_Fault => #Fault,
                   O_Warning => #Warning,
                   O_ApplicationFault => #ApplicationFault,
                   O_Brake => #Brake,
                   O_AliveBit => #AliveBit,
                   H_StatusWord1 => #"H_GBMotorEPos-MoviProPN".H_StatusWord1[1].H_Word,
                   H_StatusWord2 => #"H_GBMotorEPos-MoviProPN".H_StatusWord2[1].H_Word,
                   H_StatusWord3 => #"H_GBMotorEPos-MoviProPN".H_StatusWord3[1].H_Word,
                   H_ControlWord1 => #"H_GBMotorEPos-MoviProPN".H_ControlWord1[1].H_Word,
                   H_ControlWord2 => #"H_GBMotorEPos-MoviProPN".H_ControlWord2[1].H_Word,
                   H_SetpointPosition => #"H_GBMotorEPos-MoviProPN".H_SetpointPosition[1].H_DInt,
                   H_SetpointSpeed => #"H_GBMotorEPos-MoviProPN".H_SetPointSpeed[1].H_Int,
                   H_Acceleration => #"H_GBMotorEPos-MoviProPN".H_SetpointAcceleration[1].H_Int,
                   H_Deceleration => #"H_GBMotorEPos-MoviProPN".H_SetpointDeceleration[1].H_Int,
                   H_ActualSpeed => #"H_GBMotorEPos-MoviProPN".H_ActualSpeed[1].H_Int,
                   H_ActualPosition => #"H_GBMotorEPos-MoviProPN".H_ActualPosition[1].H_DInt,
                   H_ActualCurrentA => #"H_GBMotorEPos-MoviProPN".H_ActualCurrentA[1].H_Real,
                   "H_ActualCurrent%" => #"H_GBMotorEPos-MoviProPN".H_ActualCurrentProCent[1].H_Real,
                   H_ActualWarning => #"H_GBMotorEPos-MoviProPN".H_ActualWarning[1].H_Int,
                   H_ActualFault => #"H_GBMotorEPos-MoviProPN".H_ActualFault[1].H_Int);
   END_IF;
END_REGION

REGION Network 12: **** 8 - Outputs **** Motor turning
   #O_MotorTurning := #MotorTurning;
END_REGION

REGION Network 13: **** 8 - Outputs **** Standstill
   #O_Standstill := NOT #MotorTurning AND NOT #Brake;
END_REGION

REGION Network 14: **** 8 - Outputs **** Brake
   #O_Brake := #Brake;
END_REGION

REGION Network 15: **** 8 - Outputs **** Brake / **** 8 - Outputs **** Actual position
   IF "TRUE" THEN #O_ActualPosition := #"H_GBMotorEPos-MoviProPN".H_ActualPosition[1].H_DInt; END_IF;
END_REGION

REGION Network 16: **** 8 - Outputs **** Motor protection alarm
   // Motor protection alarm
   #O_MotorProtectionAlarm := #MotorProtectionAlarm;
END_REGION

REGION Network 17: **** 8 - Outputs **** Safety switch alarm
   // Safety switch alarm
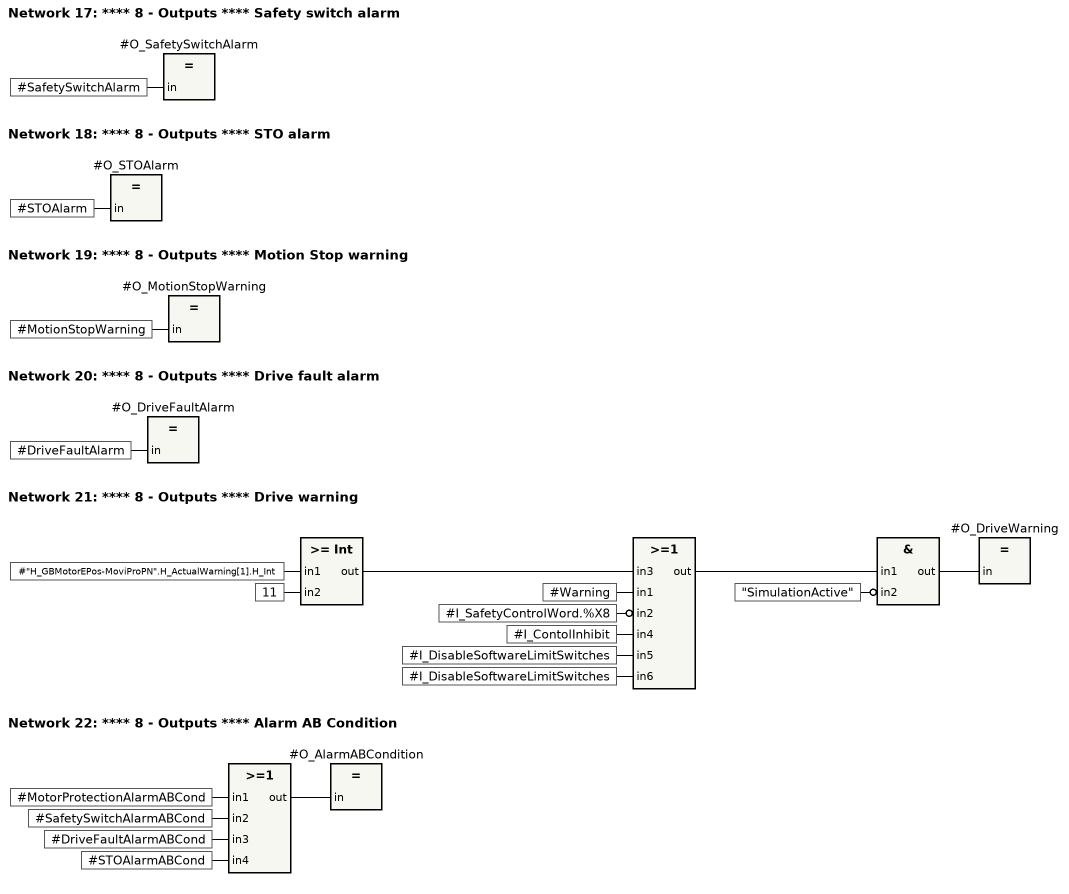
   #O_SafetySwitchAlarm := #SafetySwitchAlarm;
END_REGION

REGION Network 18: **** 8 - Outputs **** STO alarm
   #O_STOAlarm := #STOAlarm;
END_REGION

REGION Network 19: **** 8 - Outputs **** Motion Stop warning
   #O_MotionStopWarning := #MotionStopWarning;
END_REGION

REGION Network 20: **** 8 - Outputs **** Drive fault alarm
   // Drive fault
   #O_DriveFaultAlarm := #DriveFaultAlarm;
END_REGION

REGION Network 21: **** 8 - Outputs **** Drive warning
   #O_DriveWarning := ((#"H_GBMotorEPos-MoviProPN".H_ActualWarning[1].H_Int >= 11) OR #Warning OR NOT #I_SafetyControlWord.%X8 OR #I_ContolInhibit OR #I_DisableSoftwareLimitSwitches OR #I_DisableSoftwareLimitSwitches) AND NOT "SimulationActive";
END_REGION

REGION Network 22: **** 8 - Outputs **** Alarm AB Condition
   // Alarm AB Condition
   #O_AlarmABCondition := #MotorProtectionAlarmABCond OR #SafetySwitchAlarmABCond OR #DriveFaultAlarmABCond OR #STOAlarmABCond;
END_REGION
END_FUNCTION_BLOCK
